// TIA Portal project "bad_apple_hmi_test" (V16)

(* hardware
DEVICE "S71500/ET200MP station_1"  S7-1500 station
   slot 0: "Rail_0"  Rack  6ES7 590-1***0-0AA0
   slot 1: "PLC_1"  CPU 1512C-1 PN  6ES7 512-1CK01-0AB0  V2.8
      slot 3: "CPU display_1"  6ES7591-1AA00-0AA0
      slot 32768: "PROFINET interface_1"  X1
         slot 32769: "Port_1"  X1 P1
         slot 32770: "Port_2"  X1 P2
      slot 34817: "Virtual CP interface port_1"  Virtual CP interface port  Virtual CP interface port
DEVICE "HMI_1"  TP700 Comfort
   slot 0: "HMI_1"  TP700 Comfort  6AV2 124-0GC01-0AX0  16.0.0.0
   slot 1: "HMI_RT_1"  TP700 Comfort  6AV2 124-0GC01-0AX0  16.0.0.0
   slot 5: "HMI_1.IE_CP_1"  PROFINET Interface  16.0.0.0
      slot 1: "PROFINET Interface_1"  PROFINET Interface
         slot 1: "Port_1"  Port
         slot 2: "Port_2"  Port
   slot 7: "HMI_1.MPI/DP_CP_1"  MPI/DP Interface  16.0.0.0
*)

// ===== PLC "PLC_1"  CPU 1512C-1 PN =====

VAR_GLOBAL   // PLC tag table "Default tag table"
   "Clock_Byte" AT %MB10 : Byte;
   "Clock_10Hz" AT %M10.0 : Bool;
   "Clock_5Hz" AT %M10.1 : Bool;
   "Clock_2.5Hz" AT %M10.2 : Bool;
   "Clock_2Hz" AT %M10.3 : Bool;
   "Clock_1.25Hz" AT %M10.4 : Bool;
   "Clock_1Hz" AT %M10.5 : Bool;
   "Clock_0.625Hz" AT %M10.6 : Bool;
   "Clock_0.5Hz" AT %M10.7 : Bool;
   "Counter" AT %MW12 : Int;
   "Step" AT %MW14 : Int;
   "Start_hmi" AT %M16.0 : Bool;
   "Stop_hmi" AT %M16.1 : Bool;
   "Reset_hmi" AT %M16.2 : Bool;
   "yeellow" AT %Q1.5 : Bool;
   "green" AT %Q1.3 : Bool;
   "Tag_1" AT %T1 : Timer;
END_VAR

ORGANIZATION_BLOCK "Main"   // OB1, LAD, ProgramCycle
TITLE = "Main Program Sweep (Cycle)"
{ S7_Optimized_Access := 'TRUE' }
VERSION : 0.1
   VAR_INPUT
      Initial_Call : Bool;   // Initial call of this OB
      Remanence : Bool;   // =True, if remanent data are available
   END_VAR
   VAR_TEMP   // added for the SCL form of the ladder/FBD networks
      _w1 : Bool;
      _s5time1 : S5Time;
   END_VAR
BEGIN

REGION Network 1
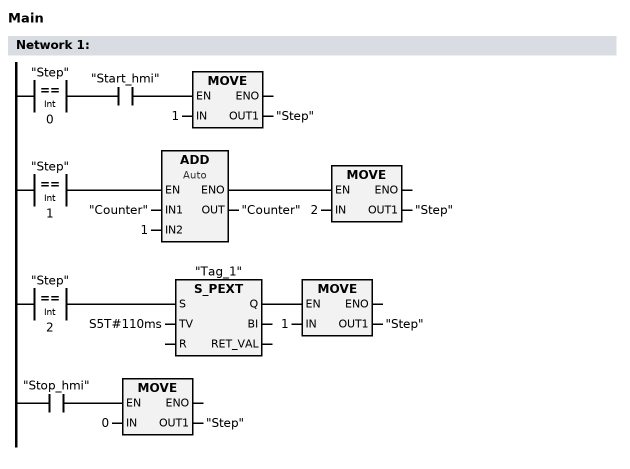
   RUNG wire#powerrail
      { S7_Templates := "SrcType := Int" } EQ_Contact(in1 := "Step", in2 := 0)
      Contact( "Start_hmi" )
      Move(in := 1, out1 => "Step")
   END_RUNG
   RUNG wire#powerrail
      { S7_Templates := "SrcType := Int" } EQ_Contact(in1 := "Step", in2 := 1)
      Add(in1 := "Counter", in2 := 1, out => "Counter")
      Move(in := 2, out1 => "Step")
   END_RUNG
   RUNG wire#powerrail
      { S7_Templates := "SrcType := Int" } EQ_Contact(in1 := "Step", in2 := 2)
      S_PEXT(T_NO := "Tag_1", TV := S5T#110ms, R :=, BI =>, RET_VAL =>)
      Move(in := 1, out1 => "Step")
   END_RUNG
   RUNG wire#powerrail
      Contact( "Stop_hmi" )
      Move(in := 0, out1 => "Step")
   END_RUNG
   // the same network as SCL:
   IF ("Step" = 0) AND "Start_hmi" THEN "Step" := 1; END_IF;
   IF "Step" = 1 THEN
       "Counter" := "Counter" + 1;
       "Step" := 2;
   END_IF;
   #_s5time1 := S_PEXT(T_NO := "Tag_1", S := "Step" = 2, TV := S5T#110ms, Q => #_w1);
   IF #_w1 THEN "Step" := 1; END_IF;
   IF "Stop_hmi" THEN "Step" := 0; END_IF;
END_REGION
END_ORGANIZATION_BLOCK

(* ===== HMI "HMI_RT_1" =====
system functions are stored by id; their names below are inferred from use
connection "HMI_Connection_1": ETHERNET, S7_1500_OMS

HMI tags "Default tag table"
   "Tag_ScreenNumber" : UInt, internal
   "Counter" : Int = PLC Counter AT %MW12, 100 ms
   "Step" : Int = PLC Step AT %MW14, 100 ms
   "Start_hmi" : Bool = PLC Start_hmi AT %M16.0, 100 ms
   "Stop_hmi" : Bool = PLC Stop_hmi AT %M16.1, 100 ms
   "Reset_hmi" : Bool = PLC Reset_hmi AT %M16.2, 100 ms

screen "Root screen" 800x424, template "Template_1"
   on GenerateScreen: SetTag("Tag_ScreenNumber", 1)
   TextField "HmiScreenItemData" at 91,26 size 640x25; Text 'Bad Apple Test 5 Frames'
   Button "Button_1" at 45,58 size 96x58; TextOff 'START'
      on Press: SetBit("Start_hmi")
      on Release: ResetBit("Stop_hmi")
   Button "Button_2" at 154,56 size 96x58; TextOff 'STOP'
      on Press: SetBit("Stop_hmi")
      on Release: SetBit("Stop_hmi")
   IOField "I/O field_1" at 45,154 size 96x32; FormatPattern s99999
      ProcessValue <- "Counter"
   TextField "Text field_1" at 53,187 size 77x23; Text 'Counter'
   Button "Button_3" at 258,161 size 192x100; TextOff 'Screen_1'
      on Click: ActivateScreen("Screen_1", 0)

Template "Template_1" 800x424
   Button "Exit" at 720,360 size 78x58; TextOff 'Exit'; PictureOff "ExitRuntime_TP700_Comfort_TR"; PictureOn "ExitRuntime_TP700_Comfort_TR"
      on Release: StopRuntime(0)
   Button "Template_Button" at 640,360 size 78x58; TextOff 'Text'
   Button "Template_Button_1" at 560,360 size 78x58; TextOff 'Text'
   Button "Template_Button_2" at 480,360 size 78x58; TextOff 'Text'
   Button "Template_Button_3" at 400,360 size 78x58; TextOff 'Text'
   Button "Template_Button_4" at 321,360 size 78x58; TextOff 'Text'
   Button "Template_Button_5" at 241,360 size 78x58; TextOff 'Text'
   Button "Template_Button_6" at 161,360 size 78x58; TextOff 'Text'
   Button "Template_Button_7" at 81,360 size 78x58; TextOff 'Text'
   Button "Start screen" at 1,360 size 78x58; TextOff 'Start screen'; PictureOff "NavigateHome_TP700_Comfort_TR"; PictureOn "NavigateHome_TP700_Comfort_TR"
      on Release: ActivateScreen("Root screen", 0)

screen "Screen_1" 800x424
   GraphicView "Graphic view_1" at 183,0 size 610x423; Picture "frame00041"
      Visibility <- "Counter"
   GraphicView "Graphic view_2" at 183,0 size 610x423; Picture "frame00042"
      Visibility <- "Counter"
   GraphicView "Graphic view_3" at 183,0 size 610x423; Picture "frame00043"
      Visibility <- "Counter"
   GraphicView "Graphic view_4" at 183,0 size 610x423; Picture "frame00044"
      Visibility <- "Counter"
   GraphicView "Graphic view_5" at 183,0 size 610x423; Picture "frame00045"
      Visibility <- "Counter"
   Button "Button_1" at 27,56 size 96x58; TextOff 'START'
      on Release: ResetBit("Stop_hmi")
      on Press: SetBit("Start_hmi")
   Button "Button_2" at 27,135 size 96x58; TextOff 'STOP'
      on Release: SetBit("Stop_hmi")
      on Press: SetBit("Stop_hmi")
   IOField "I/O field_1" at 31,217 size 96x32; FormatPattern s99999
      ProcessValue <- "Counter"
   TextField "Text field_1" at 37,252 size 77x23; Text 'Counter'
   Button "Button_3" at 0,390 size 179x32; TextOff 'Root screen'
      on Click: ActivateScreen("Root screen", 0)
*)